(* CoDeSys 2.3 export: FB_AUXILIARYSTEP.EXP *)

(* POU 4_DoorFunctions/FB_auxiliarystep, LD *)
FUNCTION_BLOCK FB_auxiliarystep
VAR_INPUT
	speedover5				:BOOL;
	pressureOK				:BOOL;
	auxstepoutward			:BOOL;
	auxstepinward			:BOOL;
	chassisVoltageOK		:BOOL;
END_VAR
VAR_OUTPUT
	auxliarystepOUTWARD	:BOOL;
END_VAR
VAR
	sr1							:SR;
END_VAR
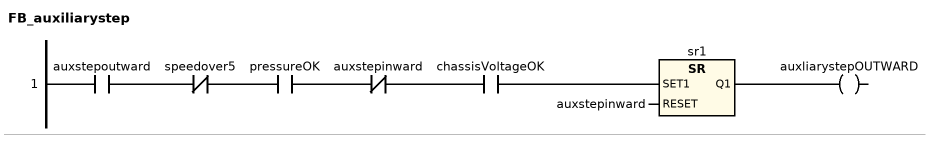
_LD_ (* Ladder Diagram *)
NETWORK 1
	[auxstepoutward] - [/speedover5] - [pressureOK] - [/auxstepinward] - [chassisVoltageOK] - sr1:SR(SET1: *, RESET: auxstepinward) --- (auxliarystepOUTWARD)
_END_LD_
(* the same logic as Structured Text *)
(* Network 1 *)
sr1(SET1 := auxstepoutward AND NOT speedover5 AND pressureOK AND NOT auxstepinward AND chassisVoltageOK, RESET := auxstepinward);
auxliarystepOUTWARD := sr1.Q1;
END_FUNCTION_BLOCK
